{attribute 'qualified_only'}
{attribute 'to_string'}
TYPE
    ErrorIDMappingLibraryTurck :
    (
        NO_ERROR := 0,
        TIME_OUT,
        FB_PARAMETER,
        CHANNEL_INACTIVE := 16#8000,
        RW_HEAD_NOT_CONNECTED,
        MEMORY_FULL,
        BLOCK_SIZE_NOT_SUPPORTED,
        LENGTH_GREATER_THEN_READ_FRAGMENT_SIZE,
        LENGTH_GREATER_THEN_WRITE_FRAGMENT_SIZE,
        PARAMETER_UNDEFINED,
        PARAMETER_OUT_OF_RANGE_OPERATING_MODE,
        PARAMETER_OUT_OF_RANGE_TAGTYPE,
        PARAMETER_OUT_OF_RANGE_CMD_REPORT_MODE,
        PARAMETER_OUT_OF_RANGE_LENGTH_REPORT_MODE,
        PARAMETER_OUT_OF_RANGE_WRITE_FRAGMENT_SIZE,
        PARAMETER_OUT_OF_RANGE_READ_FRAGMENT_SIZE,
        PARAMETER_OUT_OF_RANGE_BYPASS_TIME,
        PARAMETER_OUT_OF_RANGE_ADRESS_REPORT_MODE,
        PARAMETER_NO_RW_HEAD_SELECTED,
        COMMAND_CODE_UNKNOWN := 16#8200,
        COMMAND_NOT_SUPPORTED,
        COMMAND_NOT_SUPPORTED_FOR_HF,
        COMMAND_NOT_SUPPORTED_FOR_UHF,
        COMMAND_NOT_SUPPORTED_IN_AUTOMATIC_MODE_AND_ANTICOLLISION_MODE,
        COMMAND_NOT_SUPPORTED_IN_AUTOMATIC_MODE,
        COMMAND_NOT_SUPPORTED_OUTSIDE_AUTOMATIC_MODE,
        COMMAND_NOT_SUPPORTED_IN_ANTICOLLISON_MODE,
        COMMAND_NOT_SUPPORTED_IN_MULTI_DROP_MODE,
        COMMAND_LENGTH_OUT_OF_RANGE,
        COMMAND_ADRESS_OUT_OF_RANGE,
        COMMAND_ADRESS_PLUS_LENGTH_OUT_OF_RANGE,
        COMMAND_NO_TAG_FOUND,
        COMMAND_TIMEOUT_ELAPSED,
        COMMAND_NEXT_NOT_SIPPORTED_IN_ANTICOLLISION_MODE,
        COMMAND_SIZE_OF_UID_OUT_OF_RANGE,
        COMMAND_LENGTH_OUTSIDE_TAG_SPECS,
        COMMAND_ADDRESS_OUTSIDE_TAG_SPECS,
        COMMAND_ADRESS_PLUS_LENGTH_OUTSIDE_TAG_SPECS,
        COMMAND_MEMORY_AREA_OUT_OF_RANGE,
        COMMAND_ANTENNA_NO_OUT_OF_RANGE,
        COMMAND_TIMEOUT_VALUE_OUT_OF_RANGE,
        COMMAND_CONTINOUS_MODE_NOT_ENABLED,
        COMMAND_GROUPING_NOT_SUPPORTED_IN_HF,
        VERIFY_ERROR                := 16#801,
        COMMAND_KILL_NOT_SUCCESFULL := 16#2000,
        AUTO_TUNING_IS_ACTIVE       := 16#2200,
        TUNE_TAG_FAILED,
        PASSWORD_FUNTCTIONS_NOT_SUPPORTED_BY_TAG := 16#2500,
        PASSWORD_FUNTCTIONS_NOT_SUPPORTED_BY_RW_HEAD,
        COMMAND_ADDRESS_OUTSIDE_BLOCK_BOUNDARIES := 16#2900,
        LEN_UNDERRUN_IN_RESPONSE                 := 16#C000,
        NOT_SUPPORTED_BY_RW_HEAD_VERSION
    );
END_TYPE

(* stored: Version 1.1.0.1, ProductVersion 3.1.4024.12
   DUT ErrorIDMappingLibraryTurck: Id {7fd1ad5f-d8c4-0d6d-3083-4947fa743ed5} *)
